FUNCTION_BLOCK FB_HwRefUnistat
VAR_INPUT
END_VAR
VAR_OUTPUT
END_VAR
VAR
	SerialPort 	: REFERENCE TO FB_SerialComPort_Base;
	fbSendCmd 	: FB_Unistat_SendCmd;
	
	bPolling			: BOOL := TRUE;
	nCurrentTempIntern 	: DINT;
	nCurrentTempExtern 	: DINT;
	eState				: E_UnistatState;
	nState				: USINT;
	nStateNext			: USINT := 1;
END_VAR

IF NOT __ISVALIDREF(SerialPort) THEN
	RETURN;
END_IF
fbSendCmd.SerialPort REF= SerialPort;
IF NOT SerialPort.bIsWorking THEN
	RETURN;
END_IF

IF nState = 0 THEN
	IF bPolling THEN
		nState := nStateNext;
	END_IF
END_IF

CASE nState OF
	1:	//Status abrufen
		fbSendCmd(bExecute:= TRUE, eCommand:= E_Unitstat_Command.Get_Status);
		IF NOT fbSendCmd.bBusy THEN
			IF NOT fbSendCmd.bError THEN
				eState := fbSendCmd.nReceiveData;
			END_IF
			fbSendCmd(bExecute:= FALSE);
			nState := 0;
			nStateNext := 2;
		END_IF	

	2:	//Temp intern abrufen
		fbSendCmd(bExecute:= TRUE, eCommand:= E_Unitstat_Command.Get_TempActualIntern);
		IF NOT fbSendCmd.bBusy THEN
			IF fbSendCmd.bError THEN
				nCurrentTempIntern := 16#FFFF;
			ELSE
				nCurrentTempIntern := fbSendCmd.nReceiveData;
			END_IF
			fbSendCmd(bExecute:= FALSE);
			nState := 0;
			nStateNext := 3;
		END_IF
	3:	//Temp extern abrufen
		fbSendCmd(bExecute:= TRUE, eCommand:= E_Unitstat_Command.Get_TempActualExtern);
		IF NOT fbSendCmd.bBusy THEN
			IF fbSendCmd.bError THEN
				nCurrentTempExtern := 16#FFFF;
			ELSE
				IF fbSendCmd.nReceiveData = -1510 THEN
					nCurrentTempExtern := 16#FFFF;
				ELSE
					nCurrentTempExtern := fbSendCmd.nReceiveData;	
				END_IF
			END_IF
			fbSendCmd(bExecute:= FALSE);
			nState := 1;
			nStateNext := 1;
		END_IF
END_CASE

METHOD FB_init : BOOL
VAR_INPUT
	bInitRetains : BOOL; // if TRUE, the retain variables are initialized (warm start / cold start)
	bInCopyCode : BOOL;  // if TRUE, the instance afterwards gets moved into the copy code (online change)
	SerialPort 	: REFERENCE TO FB_SerialComPort_Base;
END_VAR
THIS^.SerialPort REF= SerialPort;
END_METHOD

PROPERTY P_bPolling : BOOL
GET
P_bPolling := bPolling;
END_GET
SET
bPolling := P_bPolling;
END_SET
END_PROPERTY

PROPERTY P_eState : E_UnistatState
GET
P_eState := eState;
END_GET
END_PROPERTY

PROPERTY P_nCurrentTempExtern : DINT
GET
P_nCurrentTempExtern := nCurrentTempExtern;
END_GET
END_PROPERTY

PROPERTY P_nCurrentTempIntern : DINT
GET
P_nCurrentTempIntern := nCurrentTempIntern;
END_GET
END_PROPERTY

PROPERTY P_SerialPort : REFERENCE TO FB_SerialComPort_Base
GET
P_SerialPort REF= SerialPort;
END_GET
END_PROPERTY

END_FUNCTION_BLOCK

(* stored: Version 1.1.0.1, ProductVersion 3.1.4024.6
   POU FB_HwRefUnistat: Id {1f3a8ac2-b2e6-4c49-959b-680e319c841a}, SpecialFunc None
   Method FB_init: Id {1f73a08f-2ff2-4e08-8f4d-0dc18f6f5e64}
   Property P_bPolling: Id {d13d508d-beeb-4fad-a4ce-076834ef14cf}
   Get Get: Id {e456d63c-5196-4245-a923-8be93098698b}
   Set Set: Id {d6d04eff-5b7a-4369-a2eb-edd357694c15}
   Property P_eState: Id {bd46d361-6428-4034-86d8-31d3303ed681}
   Get Get: Id {c96501a0-02f6-41e9-891d-452874b7b320}
   Property P_nCurrentTempExtern: Id {8a82704e-acd0-4223-965e-f51141a53834}
   Get Get: Id {6a668fbc-75c3-4c5f-84ab-d6c3be276904}
   Property P_nCurrentTempIntern: Id {c43559a4-6e4d-41e8-a347-5d499abeb97e}
   Get Get: Id {13b5494c-6c55-476e-96f5-de6d9ca9a1f2}
   Property P_SerialPort: Id {214c704f-4340-4806-bd93-a6e2ab295c46}
   Get Get: Id {263613bc-57b9-4fde-a42d-74be543a7534} *)
